// TIA Portal V21 export
FUNCTION "Dzielenie" : Void   // FC3, LAD
{ S7_Optimized_Access := 'TRUE' }
// stored: SetENOAutomatically false
BEGIN

REGION Network 1
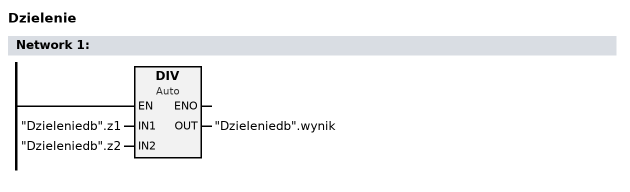
   RUNG wire#powerrail
      { S7_GenerateENO := "TRUE" } Div(in1 := "Dzieleniedb".z1, in2 := "Dzieleniedb".z2, out => "Dzieleniedb".wynik)
   END_RUNG
   // the same network as SCL:
   "Dzieleniedb".wynik := "Dzieleniedb".z1 / "Dzieleniedb".z2;
END_REGION
END_FUNCTION
